// SIMATIC S7-200 project (STEP 7-Micro/WIN), CPU 224 REL 02.01

SYMBOL_TABLE USER1
start            M0.2     // khoi dong he thong
stopp            M0.3     // dung he thong
d1               Q0.0     // den do 1
v1               Q0.1     // den vang 1
x1               Q0.2     // den xanh 1
d2               Q0.3     // den do 2
v2               Q0.4     // den vang 2
x2               Q0.5     // den xanh 2
t_1              VW10     // thoi gian den do
t_2              VW12     // thoi gian den vang
t_3              VW14     // thoi gian den xanh
t                VW18     // thoi gian tong
END_SYMBOL_TABLE

ORGANIZATION_BLOCK MAIN:OB1
TITLE=PROGRAM COMMENTS
BEGIN
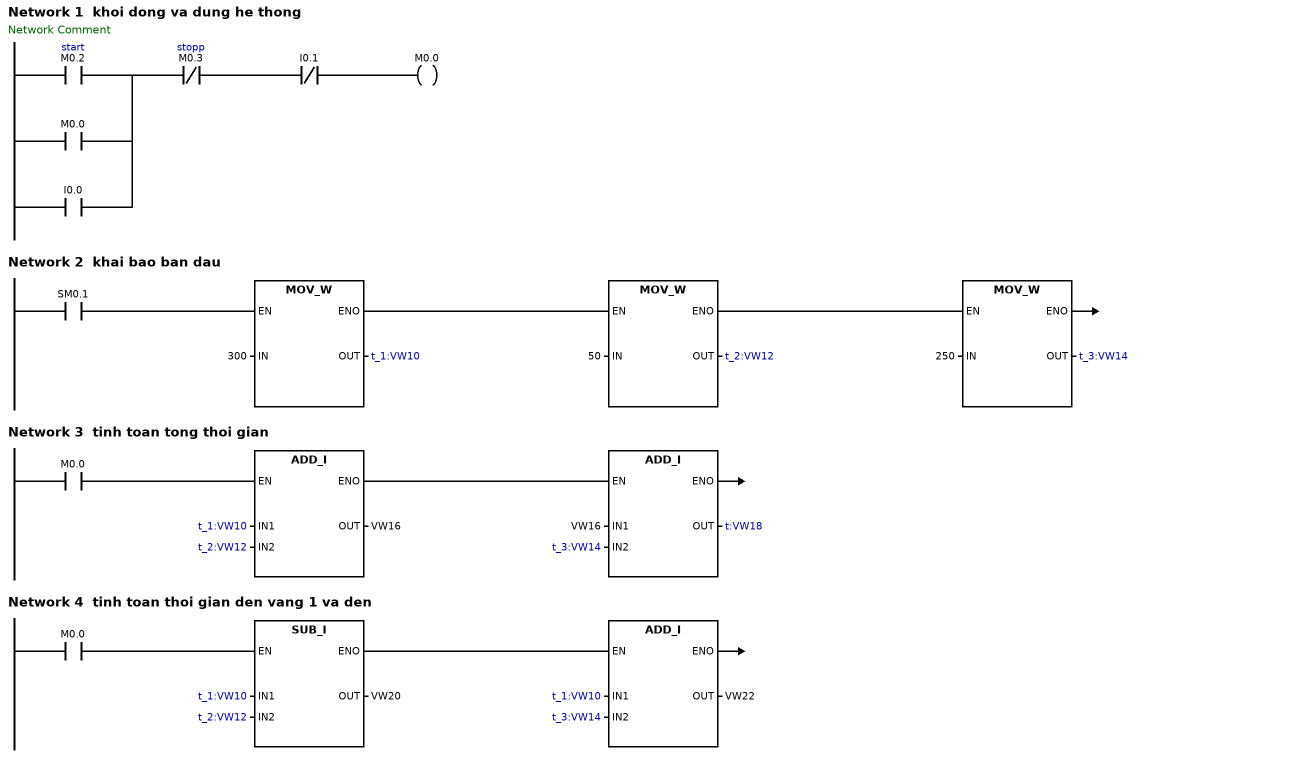
Network 1 // khoi dong va dung he thong
// Network Comment
LD     start:M0.2
O      M0.0
O      I0.0
AN     stopp:M0.3
AN     I0.1
=      M0.0
Network 2 // khai bao ban dau
LD     SM0.1
MOVW   300, t_1:VW10
AENO
MOVW   50, t_2:VW12
AENO
MOVW   250, t_3:VW14
Network 3 // tinh toan tong thoi gian
LD     M0.0
MOVW   t_1:VW10, VW16
AENO
+I     t_2:VW12, VW16
AENO
MOVW   VW16, t:VW18
+I     t_3:VW14, t:VW18
Network 4 // tinh toan thoi gian den vang 1 va den
LD     M0.0
MOVW   t_1:VW10, VW20
AENO
-I     t_2:VW12, VW20
AENO
MOVW   t_1:VW10, VW22
+I     t_3:VW14, VW22
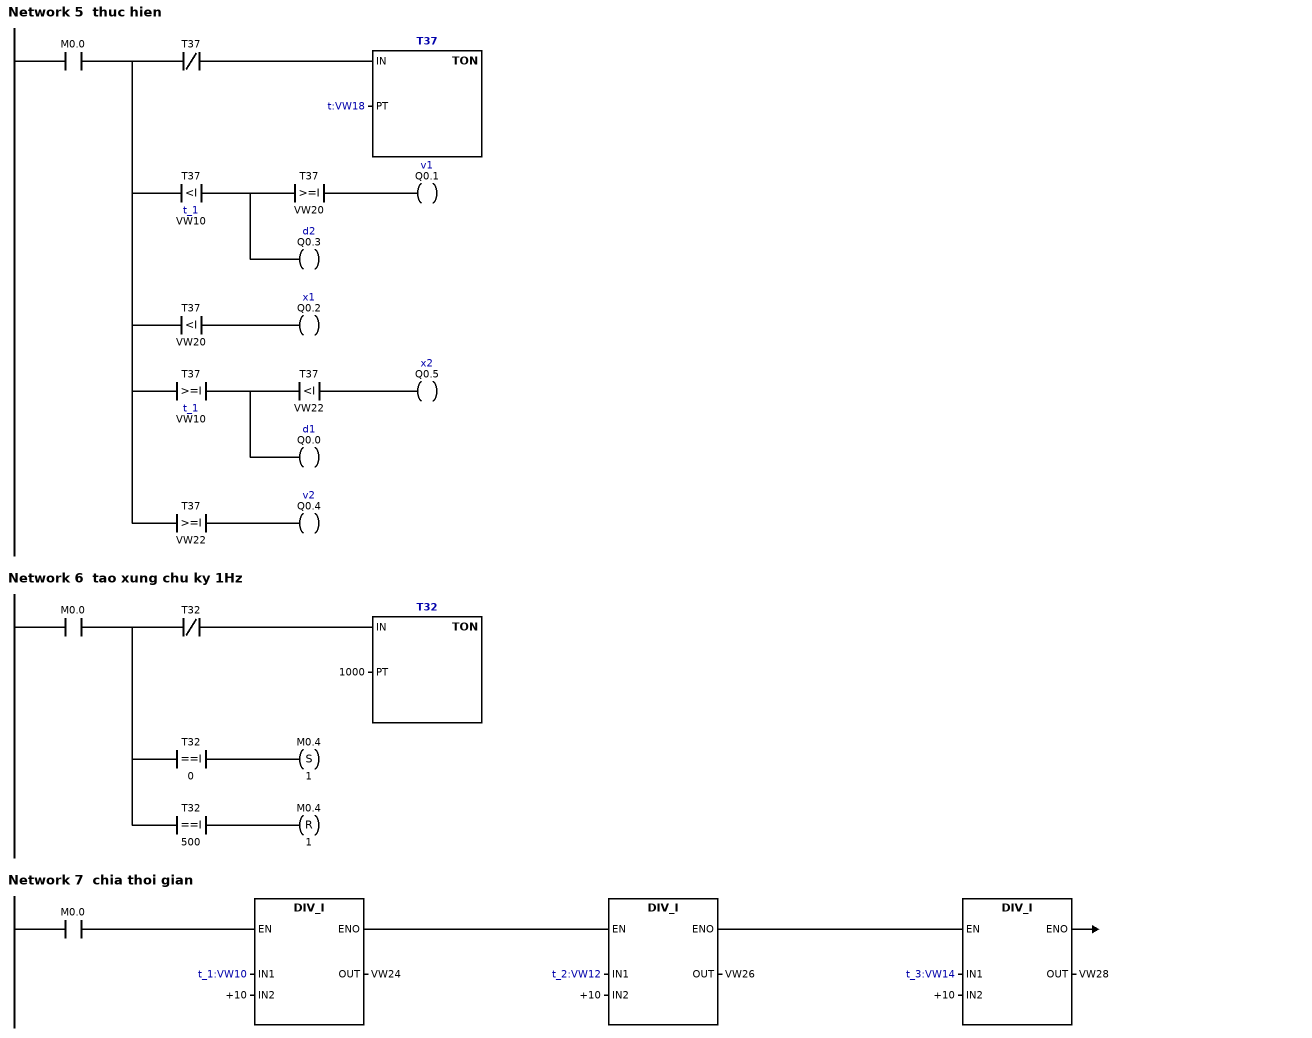
Network 5 // thuc hien 
LD     M0.0
LPS
AN     T37
TON    T37, t:VW18
LRD
AW<    T37, t_1:VW10
LPS
AW>=   T37, VW20
=      v1:Q0.1
LPP
=      d2:Q0.3
LRD
AW<    T37, VW20
=      x1:Q0.2
LRD
AW>=   T37, t_1:VW10
LPS
AW<    T37, VW22
=      x2:Q0.5
LPP
=      d1:Q0.0
LPP
AW>=   T37, VW22
=      v2:Q0.4
Network 6 // tao xung chu ky 1Hz
LD     M0.0
LPS
AN     T32
TON    T32, 1000
LRD
AW=    T32, 0
S      M0.4, 1
LPP
AW=    T32, 500
R      M0.4, 1
Network 7 // chia thoi gian
LD     M0.0
MOVW   t_1:VW10, VW24
AENO
/I     +10, VW24
AENO
MOVW   t_2:VW12, VW26
AENO
/I     +10, VW26
AENO
MOVW   t_3:VW14, VW28
/I     +10, VW28
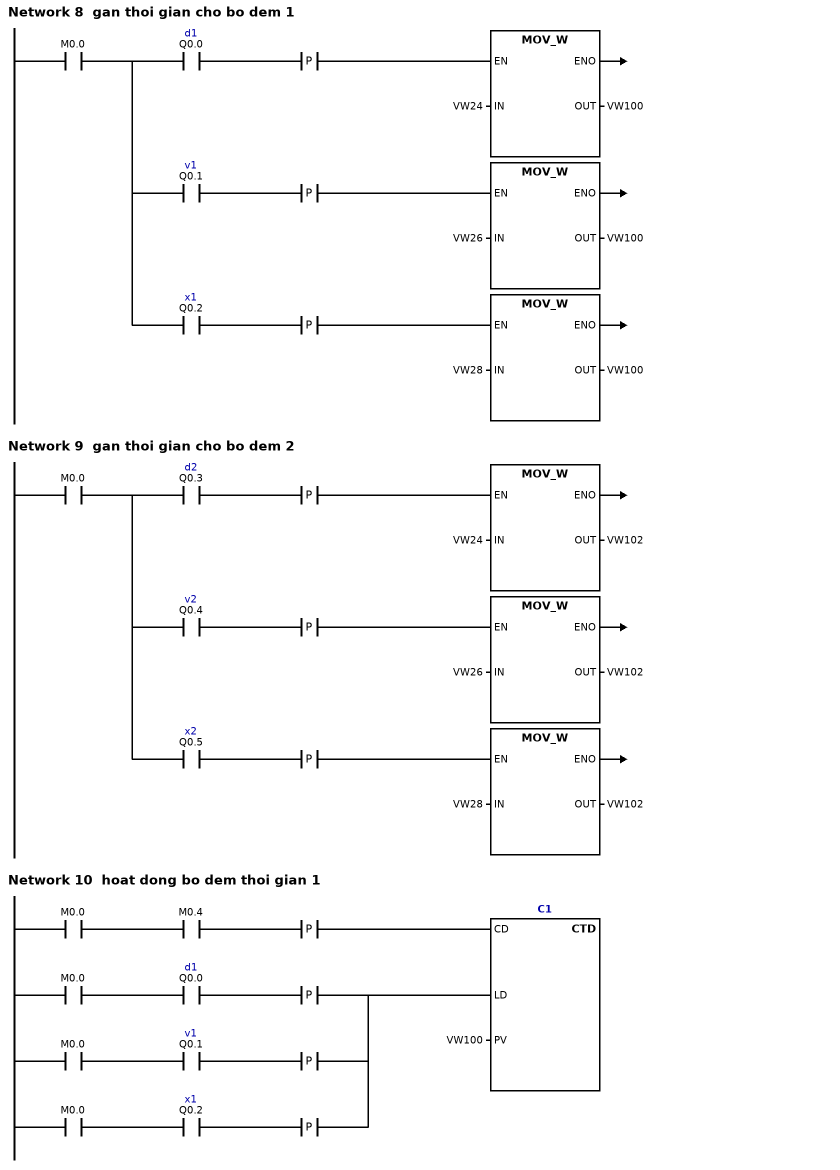
Network 8 // gan thoi gian cho bo dem 1
LD     M0.0
LPS
A      d1:Q0.0
EU
MOVW   VW24, VW100
LRD
A      v1:Q0.1
EU
MOVW   VW26, VW100
LPP
A      x1:Q0.2
EU
MOVW   VW28, VW100
Network 9 // gan thoi gian cho bo dem 2
LD     M0.0
LPS
A      d2:Q0.3
EU
MOVW   VW24, VW102
LRD
A      v2:Q0.4
EU
MOVW   VW26, VW102
LPP
A      x2:Q0.5
EU
MOVW   VW28, VW102
Network 10 // hoat dong bo dem thoi gian 1
LD     M0.0
A      M0.4
EU
LD     M0.0
A      d1:Q0.0
EU
LD     M0.0
A      v1:Q0.1
EU
OLD
LD     M0.0
A      x1:Q0.2
EU
OLD
CTD    C1, VW100
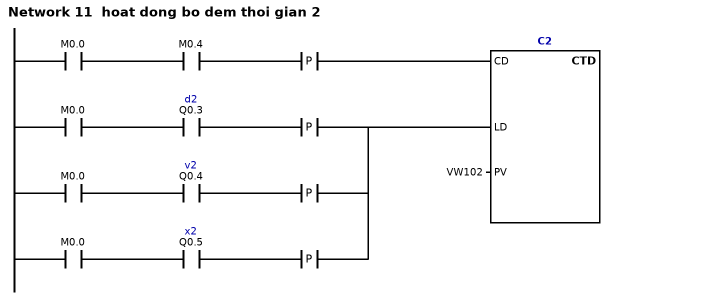
Network 11 // hoat dong bo dem thoi gian 2
LD     M0.0
A      M0.4
EU
LD     M0.0
A      d2:Q0.3
EU
LD     M0.0
A      v2:Q0.4
EU
OLD
LD     M0.0
A      x2:Q0.5
EU
OLD
CTD    C2, VW102
END_ORGANIZATION_BLOCK
